Staubli VAL3: MotionCmd.dtx

public mdesc mDesc = {leave=0, reach=0}
public num nDuration
public num nSequence
public jointRx jJointRx
